{attribute 'qualified_only'}
{attribute 'strict'}
TYPE E_Valve_State :
(
	enum_member := 0
);
END_TYPE

(* stored: Version 1.1.0.1, ProductVersion 3.1.4024.12
   DUT E_Valve_State: Id {b511b1c7-7b99-44a9-9df7-cbb7666d6bf3} *)
